TYPE DUT_HMI_09_MANUALS :
STRUCT
	PS : ARRAY[0..CNC.NUM_MAX_MANUALS_09-1] OF BOOL;
	LS : ARRAY[0..CNC.NUM_MAX_MANUALS_09-1] OF BOOL;
END_STRUCT
END_TYPE

(* stored: Version 1.1.0.1, ProductVersion 3.1.4024.13
   DUT DUT_HMI_09_MANUALS: Id {c9a71f64-971e-468a-b3bb-dcb3992928a9} *)
